FUNCTION_BLOCK FB_Int_TrigRise
VAR_INPUT
	IN:INT;
	inRequired:INT;
END_VAR
VAR_OUTPUT
	Q:BOOL;
END_VAR
VAR
	M:INT;
END_VAR
(*neste bloco funcional a saida Q e ativa durante um ciclo toda vez que IN se torna igual a inRequired*)

Q:=(IN=inRequired) AND (IN <> M);
M:=IN;

END_FUNCTION_BLOCK

(* stored: Version 1.1.0.1, ProductVersion 3.1.4024.12
   POU FB_Int_TrigRise: Id {a0d34908-8aff-4d5b-bcd1-93964bddccaa}, SpecialFunc None *)
